(*Converts data to exportable formats*)
FUNCTION_BLOCK FB_GridDataExporter EXTENDS T_NamedBase
VAR 
  // config
  _sOutPath           : T_MaxString;
  _pFbImageDeformation : POINTER TO FB_ImageDeformation;
  
  // - file handling
  bSave, bLoad        : BOOL;                   // file commands
  fbSysFile           : FB_File_Basic_SysFile;  // config file access
  
  // - json handling
  fbJson              : FB_JsonSaxWriter;       // config writer (build json string from data)
  fbJsonRd            : FB_JsonDomParser;       // config parse on read/(edit) (parse json string into data)
  jsonDoc             : STRING(nC_MaxJsonString);   // big string holding all config file

  // helper
  bInitialized, bSetup : BOOL;
  bDump               : BOOL;
  bBusy               : BOOL;
  _nSelectGrid        : UDINT;
END_VAR
VAR CONSTANT
  nC_MaxJsonString    : UDINT := 10_000;
END_VAR

// self setup -----------------------------
// - init
IF NOT bInitialized THEN Init(); RETURN; END_IF
IF NOT bSetup THEN RETURN; END_IF


IF    bSave THEN bSave := FileSave();
ELSIF bLoad THEN bLoad := FileLoad();
ELSIF bDump THEN bDump := NOT DumpGrid(); 
END_IF

METHOD PRIVATE DumpGrid : BOOL
DumpGrid := dumpJson();
END_METHOD

METHOD PRIVATE dumpJson : BOOL
VAR_OUTPUT
  nJsonSz : UDINT;
END_VAR
VAR
  i, k : UDINT := 0;
  nCamPoints : UDINT;
  sCamPoint : ST_CameraPointTbl;
  sGridPoint : ST_DeformationPointAccurate;
  nCols, nRows, nGridPoints : UDINT;
  //pTable   : POINTER TO ST_DeformationPointTbl;   // pointer to table
  sGridSettings : ST_DefGridSettings;
END_VAR
IF NOT bSetup THEN RETURN; END_IF

nCamPoints :=_pFbImageDeformation^.nAvailableCamPoints;
nGridPoints := _pFbImageDeformation^.nAvailableGridPoints;
sGridSettings := _pFbImageDeformation^.sDefGridSettings;
nCols := sGridSettings.nGridSizeX;
nRows := sGridSettings.nGridSizeY;

// build big json string ----------------------------------
fbJson.ResetDocument();
fbJson.StartObject();
// {
    fbJson.AddKey(key:='Grid');
    fbJson.StartObject();
      fbJson.AddKey(key:='NumberOfGridPoints');
      fbJson.AddUdint(value:=nGridPoints);
      fbJson.AddKey(key:='GridPoints');
      fbJson.StartArray();
      FOR i:=1 TO nRows DO
        fbJson.StartArray();
        FOR k:=1 TO nCols DO
          fbJson.StartObject();
          _pFbImageDeformation^.getDeformationPoint(nCol:=k, nRow:=i, nSel:=_nSelectGrid, sPoint=>sGridPoint, bWasSet=>);
          fbJson.AddKey(key:='col');
          fbJson.AddDint(value:=sGridPoint.col);
          fbJson.AddKey(key:='row');
          fbJson.AddDint(value:=sGridPoint.row);
          fbJson.AddKey(key:='x_ref');
          fbJson.AddLreal(value:=sGridPoint.x_ref);
          fbJson.AddKey(key:='y_ref');
          fbJson.AddLreal(value:=sGridPoint.y_ref);
          fbJson.AddKey(key:='dx');
          fbJson.AddLreal(value:=sGridPoint.dx);
          fbJson.AddKey(key:='dy');
          fbJson.AddLreal(value:=sGridPoint.dy);
          fbJson.AddKey(key:='valid');
          fbJson.AddBool(value:=sGridPoint.valid);
          fbJson.EndObject();
        END_FOR
        fbJson.EndArray();
      END_FOR
      fbJson.EndArray();
    fbJson.EndObject();
    
    
    fbJson.AddKey(key:='Cam');
    fbJson.StartObject();
      fbJson.AddKey(key:='NumberOfCamPoints');
      fbJson.AddUdint(value:=nCamPoints);
      fbJson.AddKey(key:='CamPoints');
      fbJson.StartArray();
      FOR k:=1 TO nCamPoints DO
        _pFbImageDeformation^.getCamPointX(nIdx:=k, Pn=>sCamPoint);
        fbJson.StartObject();
        fbJson.AddKey(key:='x_ref');
        fbJson.AddLreal(value:=sCamPoint.sPoint.x_ref);
        fbJson.AddKey(key:='y_ref');
        fbJson.AddLreal(value:=sCamPoint.sPoint.x_ref);
        fbJson.AddKey(key:='dx');
        fbJson.AddLreal(value:=sCamPoint.sPoint.dx);
        fbJson.AddKey(key:='dy');
        fbJson.AddLreal(value:=sCamPoint.sPoint.dy);
        fbJson.AddKey(key:='valid');
        fbJson.AddBool(value:=sCamPoint.sPoint.valid);
        fbJson.EndObject();
      END_FOR    
      fbJson.EndArray();
    fbJson.EndObject();
   
    // ]
fbJson.EndObject();
// '}'

fbJson.CopyDocument(jsonDoc, SIZEOF(jsonDoc));
// document is now in big string -----------------------------

nJsonSz := LEN2(pSTRING:=ADR(jsonDoc));
dumpJson := TRUE;
END_METHOD

(*
  Load Simulation configuration file and apply settings / modes / config to each FB_Sim.
  :return: TRUE as long busy
*)
METHOD PRIVATE FileLoad : BOOL
VAR_OUTPUT
  nError : UDINT;
END_VAR
VAR_INST
  nState : UDINT := 0;
  eof : BOOL;
  sz : UDINT := 0;
  errCode : UDINT;
END_VAR
CASE nState OF
  0:  // idle
    LogLvl(Lvl:=E_LogSeverity.Detail, 'Load file');
    IF _sOutPath <> '' THEN
      jsonDoc := '';
      nState := nState + 1; // start immediately
    ELSE
      nState := 4;   // go to parse only
    END_IF
    errCode := 0;

    
  1:  // opening file
    IF NOT fbSysFile.Open(SName:=_sOutPath, eMode:=E_FileMode.rd, bBinary:=FALSE) THEN
      IF fbSysFile.nErrId <> 0 THEN 
        errCode := fbSysFile.nErrId;
        nState := 99;
      ELSE
			  nState := nState + 1;
      END_IF
		END_IF
    
  2:  // reading file
    IF NOT fbSysFile.Read(pStr:=ADR(jsonDoc), nSize:=SIZEOF(jsonDoc), nRdBytes=>sz, bEOF=>eof) THEN
      IF fbSysFile.nErrId <> 0 THEN 
        errCode := fbSysFile.nErrId;
        nState := 99;
      ELSIF NOT eof THEN
        LogError('File could not be loaded fully');
        nState := nState + 1;
      ELSE
			  nState := nState + 1;
      END_IF
		END_IF
    
  3:  // closing file
    LogLvl(Lvl:=E_LogSeverity.Debug, Msg:=F_Concat4('Loaded file, size=', TO_STRING(sz), ' file=', _sOutPath));
    IF NOT fbSysFile.Close() THEN
      IF fbSysFile.nErrId <> 0 THEN 
        errCode := fbSysFile.nErrId;
        nState := 99;
      ELSE
			  nState := nState + 1;
      END_IF
		END_IF
    
  4:  // parsing file
    //parseJson();
    nState := nState + 1;
    
  5:  // done
    nState := 0;
    
  99: // error
    LogError(F_Concat2('Load config stopped with error', TO_STRING(errCode)));
    nState := 0;
ELSE
  ;
END_CASE

// return values
nError := errCode;
FileLoad := nState <> 0;   // busy
END_METHOD

METHOD PRIVATE FileSave : BOOL
VAR_OUTPUT
  nError : UDINT;
END_VAR
VAR_INST
  nState : UDINT := 0;
  errCode : UDINT;
  nSz : UDINT;
END_VAR
CASE nState OF
  0:  // idle
    LogLvl(Lvl:=E_LogSeverity.Detail, Msg:=F_concat2('Saving file: ', _sOutPath));
    errCode := 0;
    nState := nState + 1;
      
  1:  // parsing file
    dumpJson(nJsonSz=>nSz);
    IF _sOutPath <> '' THEN
      nState := nState + 1;
    ELSE
      nState := 5;   // done (no file to write)
    END_IF
    
  2:  // opening file
    IF NOT   fbSysFile.Open(sName:=_sOutPath, eMode:=E_FileMode.wr, bBinary:=FALSE) THEN
      IF fbSysFile.nErrId <> 0 THEN 
        errCode := fbSysFile.nErrId;
        nState := 99;
      ELSE
			  nState := nState + 1;
      END_IF
		END_IF
    
  3:  // reading file
    IF NOT fbSysFile.Write(pStr:=ADR(jsonDoc), nSize:=nSz+1) THEN
      IF fbSysFile.nErrId <> 0 THEN 
        errCode := fbSysFile.nErrId;
        nState := 99;
      ELSE
			  nState := nState + 1;
      END_IF
		END_IF
    
  4:  // closing file
    LogLvl(Lvl:=E_LogSeverity.Debug, Msg:=F_Concat2('Saved file=', _sOutPath));
    IF NOT fbSysFile.Close() THEN
      IF fbSysFile.nErrId <> 0 THEN 
        errCode := fbSysFile.nErrId;
        nState := 99;
      ELSE
			  nState := nState + 1;
      END_IF
		END_IF
    
  5:  // done
    nState := 0;
    
  99: // error
    LogError(F_Concat2('Save file stopped with error', TO_STRING(errCode)));
    nState := 0;
ELSE
  ;
END_CASE

// return values
nError := errCode;
FileSave := nState <> 0;   // busy
END_METHOD

METHOD PRIVATE Init : BOOL
LogLevel := E_LogSeverity.Info;

Init:= bInitialized := TRUE;
END_METHOD

(*
  Parse json sting into data.
  :return: TRUE on success
*)
METHOD PRIVATE parseJson : BOOL
VAR
    // parser helper variables
  bHasMember  : BOOL;
  jsonRoot    : SJsonValue;   // full doc reference
  jsonModulAry, jsonIteratorModul, jsonIteratorEndModul, jsonModul : SJsonValue;  // handling module array
  jsonModeAry, jsonIteratorMode, jsonIteratorEndMode, jsonMode : SJsonValue;      // handling mode array
  jsonProp    : SJsonValue;   // effective single entry
  arySz       : UDINT;
  
  module      : T_MaxString;
  mode        : ST_SimModeDef;
  enable      : BOOL;
  active_mode : STRING;
END_VAR
// interpret new data ------------------------------
jsonRoot := fbJsonRd.ParseDocument(sJson:=jsonDoc);
bHasMember := fbJsonRd.HasMember(jsonRoot, 'modules');
IF (bHasMember) THEN
  // moules array
  bHasMember := FALSE;
  jsonModulAry := fbJsonRd.FindMember(jsonRoot, 'modules');
  arySz := fbJsonRd.GetArraySize(jsonModulAry);
  jsonIteratorModul := fbJsonRd.ArrayBegin(jsonModulAry);
  jsonIteratorEndModul := fbJsonRd.ArrayEnd(jsonModulAry);
  WHILE jsonIteratorModul <> jsonIteratorEndModul DO
    // for each module
    jsonModul := fbJsonRd.GetArrayValue(jsonIteratorModul);
    jsonProp := fbJsonRd.FindMember(jsonModul, 'module');
    module := fbJsonRd.GetString(jsonProp);   // simulation module name
    jsonProp := fbJsonRd.FindMember(jsonModul, 'sim_enable');
    enable := fbJsonRd.GetBool(jsonProp);   // simulation enable
    jsonProp := fbJsonRd.FindMember(jsonModul, 'active_mode');
    active_mode := fbJsonRd.GetString(jsonProp);   // simulation active mode
    // mode array
    jsonModeAry := fbJsonRd.FindMember(jsonModul, 'modes');
    arySz := fbJsonRd.GetArraySize(jsonModeAry);
    jsonIteratorMode := fbJsonRd.ArrayBegin(jsonModeAry);
    jsonIteratorEndMode := fbJsonRd.ArrayEnd(jsonModeAry);
    WHILE jsonIteratorMode <> jsonIteratorEndMode DO
      // for each mode
      jsonMode := fbJsonRd.GetArrayValue(jsonIteratorMode);
      mode.aMode := fbJsonRd.GetString(jsonIteratorMode);       // get mode name
      jsonProp := fbJsonRd.FindMember(jsonMode, mode.aMode);
      fbJsonrd.CopyJson(jsonProp, mode.sCfg, SIZEOF(mode.sCfg));    // get config data (raw json)
      
      // --- setup module ---
      setupSimModule(sModule:=module, sMode:=mode, enable:=enable, active_mode:=active_mode);
      // --------------------
      
      jsonIteratorMode := fbJsonRd.NextArray(jsonIteratorMode);
		END_WHILE
    // next modules
    jsonIteratorModul := fbJsonRd.NextArray(jsonIteratorModul);
  END_WHILE
END_IF

parseJson := TRUE;    // TODO: check for parsing errors
END_METHOD

(*
  Configure the Simulation Handler.
*)
METHOD Setup : BOOL
VAR_INPUT
  sOutPath : T_MaxString;   // path to configuration .json file
  pFbImageDeformation : POINTER TO FB_ImageDeformation;
END_VAR
IF pFbImageDeformation = 0 THEN RETURN; END_IF 
IF NOT bInitialized THEN RETURN; END_IF

_sOutPath := sOutPath;
_pFbImageDeformation := pFbImageDeformation;

bSetup := TRUE;
END_METHOD

METHOD startExport
VAR_INPUT
  nSelectGrid : UDINT;
END_VAR
_nSelectGrid := nSelectGrid;
bSave := TRUE;
END_METHOD

END_FUNCTION_BLOCK

(* stored: Version 1.1.0.1, ProductVersion 3.1.4024.11
   POU FB_GridDataExporter: Id {a6e16905-996c-4000-bbd3-5d1efe3b1cb5}, SpecialFunc None
   Method DumpGrid: Id {de6113b8-c508-4943-a855-5bc858b3b061}
   Method dumpJson: Id {97cfe1c3-c8ec-4fe7-b0f0-77e52207b625}
   Method FileLoad: Id {4cd360ab-51fe-4f58-a31a-78f496b6e5e6}
   Method FileSave: Id {163aa65e-e284-4ad9-ba70-5d4737ab8950}
   Method Init: Id {0b3b4c19-d57a-460d-a755-c549681d340e}
   Method parseJson: Id {1f3da447-b504-4923-bfa9-b2d2ec7f6cf1}
   Method Setup: Id {476912bc-26a3-4d6c-8bd3-023a45209de1}
   Method startExport: Id {d8940ba5-d237-4a7b-aef8-04b7114250d0} *)
